FUNCTION_BLOCK "ST10_Stopper_FB"
VAR
  FB_Stopper_Instance : Array[1..3] of "FB_Stopper";
END_VAR
BEGIN
  // Původní jazyk: LAD
  // Zdroj XML: EXPORT/Program blocks/OP010/10_Device/06_Stopper/ST10_Stopper_FB.xml
  // --- LAD/FBD → SCL (orientační převod, jen pro revizi) ---
  // Network 1
  // --- Poznámky / omezení převodu ---
  // Síť obsahuje nepodporované prvky (ponecháno jen jako komentář): O(1)
  // Network 2
  // --- Poznámky / omezení převodu ---
  // Síť obsahuje nepodporované prvky (ponecháno jen jako komentář): O(1)
  // Network 3
  // --- Poznámky / omezení převodu ---
  // Síť obsahuje nepodporované prvky (ponecháno jen jako komentář): O(1)
END_FUNCTION_BLOCK
